// TIA Portal V19 export
DATA_BLOCK "Pu_CM05.GP11_DB"   // DB1011
// stored: AutoNumber false, InstanceOfName Pu_CM05.GP11, InstanceOfType FB
"Pu_CM05.GP11"
   // VAR RETAIN
   //    In { ExternalVisible := 'False'; ExternalWritable := 'False'} : Struct
   //       NotHalt : Bool;
   //       MSS_ok : Bool;
   //       Auto : Bool;
   //       Ein : Bool;
   //       GW_p : Bool;
   //       "Niv_Uel_CM05.BL05" : Bool;
   //       "Niv_max_CM05.BL01" : Bool;
   //       "Niv_min_CM05.BL02" : Bool;
   //       "Niv_TLS_CM05.BL03" : Bool;
   //       AWA_ok : Bool;
   //       Frg_AWA : Bool;
   //       "SRM_CM05.QM61_auf" : Bool;
   //       "SRM_CM05.QM61_zu" : Bool;
   //       "SRM_CM05.QM64_auf" : Bool;
   //       "SRM_CM05.QM64_zu" : Bool;
   //       Betriebsart : USInt;
   //       Druck_Pumpe { ExternalAccessible := 'False'} : Real;
   //    END_STRUCT;
   //    Param { ExternalVisible := 'False'; ExternalWritable := 'False'} : Struct
   //       Spülzeit : Time;
   //       DT_Druckaufbau { ExternalAccessible := 'False'} : Time;
   //       DT_Testzeit { ExternalAccessible := 'False'} : Time;
   //       SW_Drucktest { ExternalAccessible := 'False'} : Real;
   //    END_STRUCT;
   //    Zst : Struct
   //       Niveau : USInt;
   //       Status_GP11 : USInt;
   //       Status_DT { ExternalAccessible := 'False'; ExternalVisible := 'False'; ExternalWritable := 'False'} : USInt;
   //       Restzeit_Spülen : Time;
   //       Restzeit_DT { ExternalAccessible := 'False'; ExternalVisible := 'False'; ExternalWritable := 'False'} : Time;
   //       "TON_CM05.QM62_auf" : Bool;
   //       Spuelen : Bool;
   //       Zeit_laeuft { ExternalAccessible := 'False'; ExternalVisible := 'False'; ExternalWritable := 'False'} : Bool;
   //       Spuelen_aktiv : Bool;
   //       Drucktest_aktiv : Bool;
   //       Drucktest_ok { ExternalAccessible := 'False'; ExternalVisible := 'False'; ExternalWritable := 'False'} : Bool;
   //       Bedienung_erlaubt { ExternalAccessible := 'False'; ExternalVisible := 'False'; ExternalWritable := 'False'} : Bool;
   //    END_STRUCT;
   //    Mld { ExternalVisible := 'False'; ExternalWritable := 'False'} : Struct
   //       MSS : Bool;
   //       "TLS_CM05.BL03" : Bool;
   //       "Uel_CM05.BL05" : Bool;
   //       AWA_niO : Bool;
   //       keine_Frg_AWA : Bool;
   //       Niv_Sensorfehler : Bool;
   //       GW_p : Bool;
   //       n_Auto : Bool;
   //       TO_Druckaufbau { ExternalAccessible := 'False'} : Bool;
   //       Drucktest_ok { ExternalAccessible := 'False'} : Bool;
   //       DT_Fehler { ExternalAccessible := 'False'} : Bool;
   //       Pu_Spuelen_Fertig { ExternalAccessible := 'False'} : Bool;
   //    END_STRUCT;
   //    Out { ExternalVisible := 'False'; ExternalWritable := 'False'} : Struct
   //       GP11_Ein : Bool;
   //       QM61 : Bool;
   //       QM62 : Bool;
   //       QM63 : Bool;
   //       QM64 : Bool;
   //    END_STRUCT;
   // END_VAR
   // VAR
   //    IEC_Timer : Struct
   //       "CM05.QM62_auf" { ExternalAccessible := 'False'; ExternalVisible := 'False'; ExternalWritable := 'False'; S7_SetPoint := 'True'} : TON_TIME;
   //       Spülen { S7_SetPoint := 'True'} : TP_TIME;
   //       GW_p { S7_SetPoint := 'True'} : TON_TIME;
   //       Drucktest { ExternalAccessible := 'False'; ExternalVisible := 'False'; ExternalWritable := 'False'; S7_SetPoint := 'True'} : TP_TIME;
   //       TO_Druckaufbau { ExternalAccessible := 'False'; ExternalVisible := 'False'; ExternalWritable := 'False'; S7_SetPoint := 'True'} : TON_TIME;
   //       QM63 { S7_SetPoint := 'True'} : TOF_TIME;
   //    END_STRUCT;
   //    R_TRIG_Hand_EIN { S7_SetPoint := 'True'} : R_TRIG;
   // END_VAR
BEGIN
END_DATA_BLOCK
